(* IEC 61131-3 sources: Industry-PLC-LLM/data/PLCBEAD_repo/PLCBEAD_PLCEmbed-main/PLC-BEAD/Source/GEB/DIFFER, 1 file *)

(* ---- DIFFER.ST ---- *)
FUNCTION DIFFER:BOOL
	VAR_INPUT
		IN1 :	REAL;
		IN2 :	REAL;
		X :	REAL;
	END_VAR

	DIFFER := ABS(IN1 - IN2) > X;
END_FUNCTION

PROGRAM program0
  VAR
    LocalVar0 : REAL;
	LocalVaR1  : REAL;
	LocalVaR2 : REAL;
	LocalOUT  : BOOL;
  END_VAR
  	LocalOUT := DIFFER(LocalVar0, LocalVaR1 , LocalVaR2);
END_PROGRAM
